PROGRAM P_Joy
VAR
END_VAR

XboxControl.joyLeft := INT_TO_LREAL(XboxControl.controller.LeftJoystickX)/32767.0;

END_PROGRAM

(* stored: Version 1.1.0.1, ProductVersion 3.1.4024.9
   POU P_Joy: Id {5aaf6033-864c-4c13-9a1e-c92eedd8448a}, SpecialFunc None *)
